FUNCTION_BLOCK StartAtMainTask EXTENDS TcoMitsubishiRoboticsTask

IF Execute() THEN
    _blink(inOnTime := T#500MS, inOffTime := T#500MS);

    IF _progress = 0 THEN
        IF NOT __ISVALIDREF(inoControl) THEN
            _varInfo := __VARINFO(inoControl);
            Messenger.Programming(_sb.Clear().Append('<#Invalid reference: #>').Append(_varInfo.Symbol).ToString()).Pin();
        ELSIF NOT __ISVALIDREF(inoConfig) THEN
            _varInfo := __VARINFO(inoConfig);
            Messenger.Programming(_sb.Clear().Append('<#Invalid reference: #>').Append(_varInfo.Symbol).ToString()).Pin();
        ELSIF NOT __ISVALIDREF(inoStatus) THEN
            _varInfo := __VARINFO(inoStatus);
            Messenger.Programming(_sb.Clear().Append('<#Invalid reference: #>').Append(_varInfo.Symbol).ToString()).Pin();
        ELSE
            _progress := _progress + 1;
        END_IF
    END_IF

    IF _progress = 1 THEN
        inoControl.AutoEnable := TRUE;
        _varInfo := __VARINFO(inoStatus.State.AutoEnable);

        THIS^.Messenger.OnCondition(_infoTimer.Q AND NOT inoStatus.State.AutoEnable)
            .Warning(_sb.Clear().Append('<#Waiting for Auto signal! #>').Append(_varInfo.Symbol).ToString());

        IF inoStatus.State.AutoEnable THEN
            _progress := _progress + 1;
        END_IF;
    END_IF;

    IF _progress = 2 THEN
        inoControl.OperationEnable := TRUE;
        _varInfo := __VARINFO(inoStatus.State.OperationEnable);

        THIS^.Messenger.OnCondition(_infoTimer.Q AND NOT inoStatus.State.OperationEnable)
            .Warning(_sb.Clear().Append('<#Waiting for Operation enable signal! #>').Append(_varInfo.Symbol).ToString());

        IF inoStatus.State.OperationEnable THEN
            _progress := _progress + 1;
        END_IF;
    END_IF;

    IF _progress = 3 THEN
        Messenger.Debug('<#Robot Error Reset#>');
        inoControl.ErrorReset := inoStatus.State.ErrorReset AND _blink.outQ;

        IF NOT inoStatus.State.ErrorReset THEN
            inoControl.ErrorReset := FALSE;
            _progress := _progress + 1;
        END_IF
    END_IF;

    IF _progress = 4 THEN
        Messenger.Debug('<#Robot Emergency Stop Reset#>');
        inoControl.ErrorReset := inoStatus.State.EmergencyError AND _blink.outQ;

        IF NOT inoStatus.State.EmergencyError THEN
            inoControl.ErrorReset := FALSE;
            _progress := _progress + 1;
        END_IF
    END_IF;

    IF _progress = 5 THEN
        inoControl.ProgramReset := _blink.outQ;
        _varInfo := __VARINFO(inoStatus.State.ProgramReset);

        THIS^.Messenger.OnCondition(_infoTimer.Q AND NOT inoStatus.State.ProgramReset)
            .Warning(_sb.Clear().Append('<#Waiting program reset changed! #>').Append(_varInfo.Symbol).ToString());

        IF inoStatus.State.ProgramReset THEN
            inoControl.ProgramReset := FALSE;
            DoneWhen(inoStatus.State.ProgramReset);
        END_IF
    END_IF

    CallTimers(TRUE);
    THIS^.ThrowWhen(_errorTimer.Q);
END_IF;

IF THIS^.Error AND NOT _errorMessage.Pinned THEN
    THIS^.Restore();
END_IF

METHOD PUBLIC FB_init : BOOL
VAR_INPUT
    bInitRetains : BOOL; // if TRUE, the retain variables are initialized (warm start / cold start)
    bInCopyCode : BOOL; // if TRUE, the instance afterwards gets moved into the copy code (online change)
    ParentObject : ITcoObject;
END_VAR
END_METHOD

(*~
    <docu>
        <summary>
            Executes when task is aborted.
        </summary>
    </docu>
~*)
METHOD PROTECTED OnAbort
IF __ISVALIDREF(inoStatus) THEN
    THIS^.inoStatus.ActionDescription := '<#Start at Main was aborted, while not yet completed!#>';
END_IF;
END_METHOD

(*~
    <docu>
        <summary>
            Executes when task reaches the ```Done``` state .
        </summary>
    </docu>
~*)
METHOD PROTECTED OnDone
IF __ISVALIDREF(inoStatus) THEN
    THIS^.inoStatus.ActionDescription := '<#Start at Main was completed successfully.#>';
END_IF;

_progress := 0;
END_METHOD

(*~
    <docu>
        <summary>
            Executes when task reaches the ```Error``` state.
            <para>
                Do not confuse with <see cref="PlcDocu.TcoCore.TcoTask.WhileError()"/>, that is called cyclically until '''Error''' state is left.
            </para>
        </summary>
    </docu>
~*)
METHOD PROTECTED OnError
VAR
    description : STRING;
END_VAR
description := '<#Start at Main finished with error.#>';

IF __ISVALIDREF(inoStatus) THEN
    THIS^.inoStatus.ActionDescription := description;
END_IF;

THIS^._errorMessage.Error(_sb.Clear().Append(description).Append(' To restore acknowledge this alarm.').ToString()).Pin();
END_METHOD

METHOD PROTECTED OnStart
IF __ISVALIDREF(inoStatus) THEN
    THIS^.inoStatus.ActionDescription := '<#Start at Main started.#>';
END_IF;
END_METHOD

(*~
    <docu>
        <summary>
            Restores this instance to the Ready state. Can be called explicitly or from within one of the restore mechanisms.
            <para>
                See also <see cref="PlcDocu.TcoCore.TcoTask.AutoRestorable()"/>
            </para>
        </summary>
    </docu>
~*)
METHOD Restore : ITcoRestorable
SUPER^.Restore();
END_METHOD

END_FUNCTION_BLOCK

(* stored: Version 1.1.0.1, ProductVersion 3.1.4024.12
   POU StartAtMainTask: Id {9f626e70-6917-0906-0392-888f2e17689a}, SpecialFunc None
   Method FB_init: Id {46dce108-63c7-0971-07a8-26936ff0d54d}
   Method OnAbort: Id {fdcb8fea-12c7-091b-0d96-a87e947aaccc}
   Method OnDone: Id {d55cd1ac-5d06-0b09-12d7-70759219f1ae}
   Method OnError: Id {1d43d108-69af-0871-0f73-74bdd96a5cd6}
   Method OnStart: Id {f1a6edc0-aa90-06d6-2a38-0a8926fcea6d}
   Method Restore: Id {71b9f3a4-9089-0e2d-303a-b64fe1c7d462} *)
